FUNCTION_BLOCK Least_gate_element
VAR_INPUT
	Enforce:BOOL;
	Enforce_in_rope_cap:BOOL;
	Allowed_speed:REAL;
	Description:STRING[32];
END_VAR
VAR_OUTPUT
END_VAR
VAR_IN_OUT
	Least_gate_data:dut_Least_gate;
END_VAR
VAR
END_VAR

Least_gate_element_m();

METHOD Least_gate_element_m
VAR_INPUT
END_VAR
VAR_INST // added by the converter: edge detectors and wires of the graphical bodies
    _w1, _w4, _w5 : BOOL;
    _w2, _w3 : ANY;
    _w6 : REAL;
END_VAR
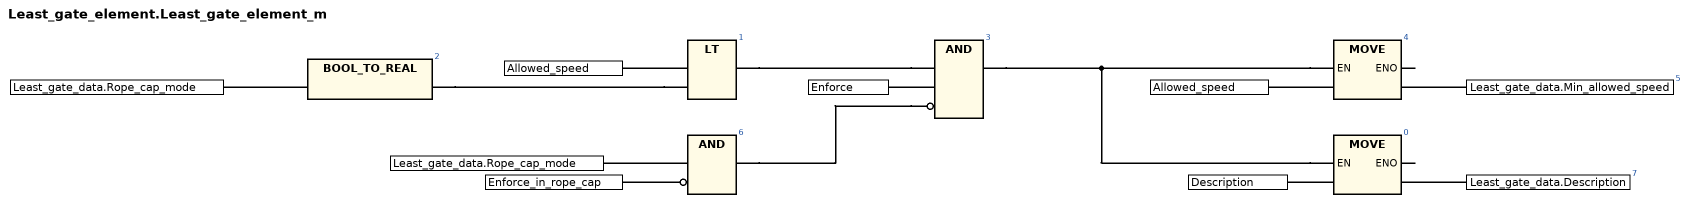
IF _w1 THEN _w2 := Description; END_IF
_w4 := Allowed_speed < _w3;
_w3 := BOOL_TO_REAL(Least_gate_data.Rope_cap_mode);
_w1 := _w4 AND Enforce AND NOT _w5;
IF _w1 THEN _w6 := Allowed_speed; END_IF
Least_gate_data.Min_allowed_speed := _w6;
_w5 := Least_gate_data.Rope_cap_mode AND NOT Enforce_in_rope_cap;
Least_gate_data.Description := _w2;
END_METHOD

END_FUNCTION_BLOCK

(* stored: Version 1.1.0.1, ProductVersion 3.1.4024.0
   POU Least_gate_element: Id {fa2e3ebe-5cbe-40bb-9103-e3031cea6602}, SpecialFunc None
   Method Least_gate_element_m: Id {5e4cbec7-f44e-4a81-b6cc-b7c86861d6cb} *)
